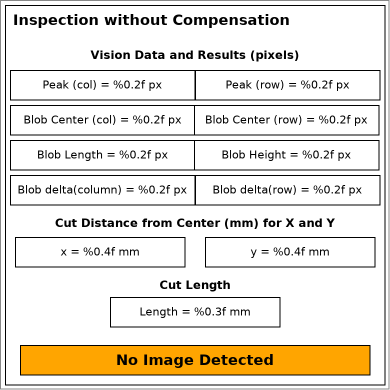
VISUALIZATION Manual_Camera_Inspection_Raw  // 390x390
    Rectangle (20,345 350x30), "PASSED", invisible if: NOT MAIN.bPassed
    Rectangle (20,345 350x30), "FAILED", invisible if: NOT MAIN.bFailed
    Rectangle (5,5 380x380)
    Label (10,5 297x30), "Inspection without Compensation"
    Rectangle (10,70 185x30), "Peak (col) = %0.2f px", text variable: MAIN.fbSlitter.Camera._columnPeak
    Rectangle (195,70 185x30), "Peak (row) = %0.2f px", text variable: MAIN.fbSlitter.Camera._rowPeak
    Rectangle (10,105 185x30), "Blob Center (col) = %0.2f px", text variable: MAIN.fbSlitter.Camera.CameraData.Results.LocationInX
    Rectangle (194,105 185x30), "Blob Center (row) = %0.2f px", text variable: MAIN.fbSlitter.Camera.CameraData.Results.LocationInY
    Rectangle (10,175 185x30), "Blob delta(column) = %0.2f px", text variable: MAIN.fbSlitter.Camera.DeltaXpx
    Rectangle (195,175 185x30), "Blob delta(row) = %0.2f px", text variable: MAIN.fbSlitter.Camera.DeltaYpx
    Rectangle (15,237 170x30), "x = %0.4f mm", text variable: MAIN.fbSlitter.Camera.DeltaXmm
    Rectangle (205,237 170x30), "y = %0.4f mm", text variable: MAIN.fbSlitter.Camera.DeltaYmm
    Label (0,208 390x30), "Cut Distance from Center (mm) for X and Y"
    Rectangle (110,297 170x30), "Length = %0.3f mm", text variable: MAIN.fbSlitter.Camera.CutLength
    Label (0,40 390x30), "Vision Data and Results (pixels)"
    Rectangle (10,140 185x30), "Blob Length = %0.2f px", text variable: MAIN.fbSlitter.Camera.CameraData.Results.WidthMeasurement
    Rectangle (194,140 185x30), "Blob Height = %0.2f px", text variable: MAIN.fbSlitter.Camera.CameraData.Results.HeightMeasurement
    Label (0,270 390x30), "Cut Length"
    Rectangle (20,345 350x30), "Processing", invisible if: NOT MAIN.bProcessing
    Rectangle (20,345 350x30), "No Image Detected", invisible if: NOT MAIN.bNoDetect
END_VISUALIZATION

(* stored: Version 1.1.0.1, ProductVersion 3.1.4024.3
   Visu Manual_Camera_Inspection_Raw: Id {e1f0ecad-66fb-4397-934b-48606ad41de2} *)
